PROGRAM prg_Teleruptor
VAR
END_VAR

END_PROGRAM

(* stored: Version 1.1.0.1, ProductVersion 3.1.4024.15
   POU prg_Teleruptor: Id {81aa6041-588d-4d22-ae97-814c8e821228}, SpecialFunc None *)
